// TIA Portal V16 export
// export: Created 2023-03-29T11:04:41.3161846Z, ExportSetting WithDefaults, DisplayName Totally Integrated Automation Portal, DisplayVersion V16 Update 6, DisplayName TIA Portal Version Control Interface, DisplayVersion V16 Update 2, DisplayName TIA Portal Openness, DisplayVersion V16 Update 6, DisplayName STEP 7 Professional, DisplayVersion V16 Update 6, DisplayName STEP 7 Safety, DisplayVersion V16, DisplayName WinCC Advanced, DisplayVersion V16 Update 6
DATA_BLOCK "dbTags_master_MPP04_1"   // DB38
{ S7_Optimized_Access := 'FALSE' }
VERSION : 0.1
// stored: AutoNumber true, DBAccessibleFromOPCUA true, IsOnlyStoredInLoadMemory false, IsWriteProtectedInAS false
   VAR
      "step" : USInt := 1;
      edge : Bool := false;
      modbusCommLoad { S7_SetPoint := 'True'} : "typeModbusCommLoad";
      modbusMaster { S7_SetPoint := 'True'} : "typeModbusMaster";
   END_VAR
BEGIN
END_DATA_BLOCK
